ADAPTER IFeedRequest (* Adapter Interface *)
  (* Standard: 61499-1 *)
  (* Version 0.0, 14/09/2026 *)
  PACKAGE Hidryco.HidrycoLib;
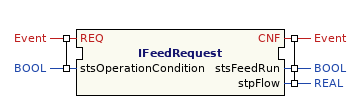
  EVENT_INPUT
    REQ WITH stsOperationCondition; (* Request from Socket *)
  END_EVENT
  EVENT_OUTPUT
    CNF WITH stsFeedRun, stpFlow; (* Confirmation from Plug *)
  END_EVENT
  VAR_INPUT
    stsOperationCondition : BOOL; (* Request Data from Socket *)
  END_VAR
  VAR_OUTPUT
    stsFeedRun : BOOL; (* Confirmation Data from Plug *)
    stpFlow : REAL; (* Indication Data from Plug *)
  END_VAR
  SERVICE SOCKET/PLUG
    SEQUENCE request_confirm
      SOCKET.REQ(stsOperationCondition) -> PLUG.REQ(stsOperationCondition);
      PLUG.CNF(stsFeedRun) -> SOCKET.CNF(stsFeedRun);
    END_SEQUENCE
    SEQUENCE indication_response
      PLUG.IND(stpFlow) -> SOCKET.IND(stpFlow);
      SOCKET.RSP(RSPD) -> PLUG.RSP(RSPD);
    END_SEQUENCE
  END_SERVICE
END_ADAPTER
